FUNCTION_BLOCK FB_ValveTrigger
VAR_INPUT
	openCommand : BOOL;
END_VAR
VAR_OUTPUT
	buttonCommand : BOOL;
	isOpen : BOOL;
END_VAR
VAR
	RTRIG_OpenCommand : R_TRIG;
	FTRIG_OpenCommand : F_TRIG;
	TON_ResetButton : TON;
	prevState : BOOL;
END_VAR


RTRIG_OpenCommand(CLK := openCommand);
FTRIG_OpenCommand(CLK := openCommand);

IF RTRIG_OpenCommand.q OR FTRIG_OpenCommand.q THEN
	isOpen := NOT isOpen;
END_IF

buttonCommand := isOpen <> prevState;

TON_ResetButton(IN := isOpen <> prevState, PT := T#100MS);
IF TON_ResetButton.q THEN
	buttonCommand := FALSE;
	prevState := isOpen;
END_IF

END_FUNCTION_BLOCK

(* stored: Version 1.1.0.1, ProductVersion 3.1.4024.9
   POU FB_ValveTrigger: Id {d21c66e5-bf67-4754-af17-31e8688193c8}, SpecialFunc None *)
